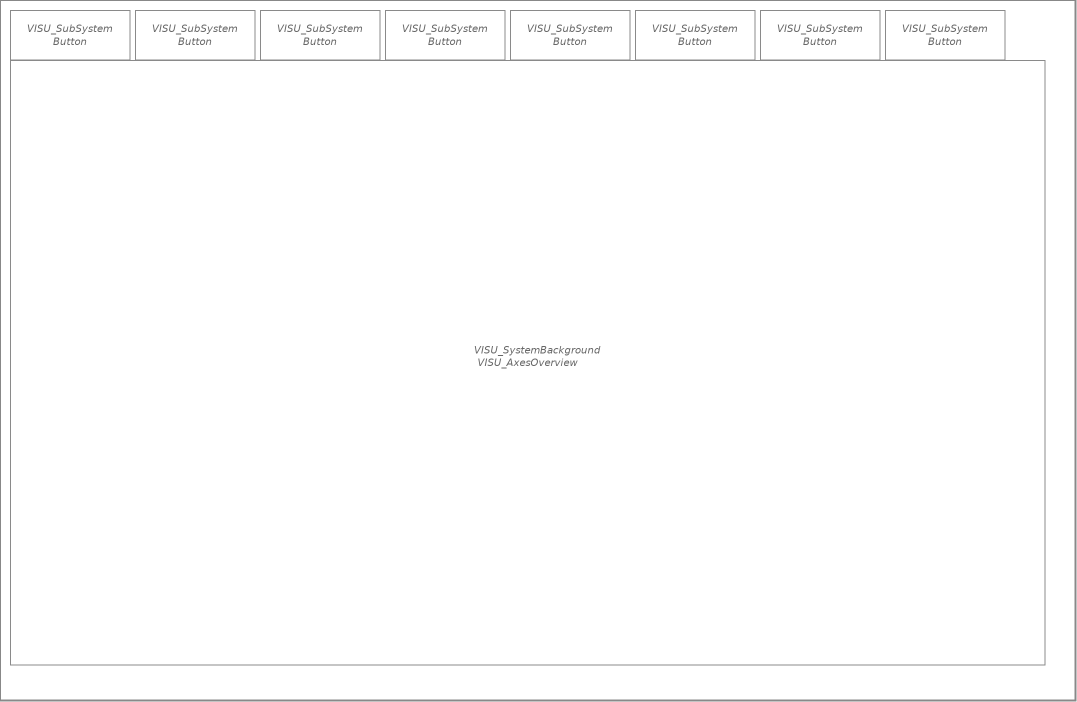
VISUALIZATION VISU_Axes  // 1077x702
VAR_IN_OUT
	ref : Axes;
    widget : AxesWidget;
END_VAR
    Frame (0,0 1075x700)
        shows VISU_SystemBackground(color := widget.actualStatus.color)
    Frame (10,60 1035x605)
        shows VISU_AxesOverview(ref := ref, widget := widget)
        shows VISU_AxesManual(ref := ref, widget := widget.manual)
        shows VISU_AxesAxes(ref := ref, widget := widget.axes)
        shows VISU_AxesTarget(ref := ref, widget := widget)
        shows VISU_AxesPointingModelsSetup(ref := ref.parts.tpoint, widget := widget.tpoint)
        shows VISU_AxesAdvanced(ref := ref, widget := widget)
        shows VISU_AxesIO(ref := ref.parts.io, widget := widget.io)
        shows VISU_AxesConfig(editable := ref.editableConfig, active := ref.config, mgr := ref.parts.configManager, mgrWidget := widget.configManager, axesWidget := widget)
        p701045219: ref.editableConfig
        p2690442461: ref.config
        p942769723: ref.parts.configManager
        p2963374678: widget.configManager
        p459268616: widget
        p4094514409: widget
        p1371549466: ref.editableConfig
        p1340763843: ref.config
        p2803088772: widget
        p2427492753: ref.parts.aziDrive
        p1656878407: ref.parts.ablDrive
        p2190985393: ref.parts.eleDrive
    Frame (10,10 120x50)
        shows VISU_SubSystemButton(widget := widget.button_overview)
        OnMouseClick: FrameSelectionChange Selection=SelectedFrame=b1e9e4b0-bf3d-440f-90c5-cb513105ccf1, GlobSel=AssignType=Directly, SelType=Locally
        OnMouseClick: execute { widget.activeTab := AxesTabs.OVERVIEW; }
    Frame (635,10 120x50)
        shows VISU_SubSystemButton(widget := widget.button_advanced)
        OnMouseClick: FrameSelectionChange Selection=SelectedFrame=b1e9e4b0-bf3d-440f-90c5-cb513105ccf1, Selection=5, GlobSel=AssignType=Directly, SelType=Locally
        OnMouseClick: execute { widget.activeTab := AxesTabs.ADVANCED; }
    Frame (760,10 120x50)
        shows VISU_SubSystemButton(widget := widget.button_io)
        OnMouseClick: FrameSelectionChange Selection=SelectedFrame=b1e9e4b0-bf3d-440f-90c5-cb513105ccf1, Selection=6, GlobSel=AssignType=Directly, SelType=Locally
        OnMouseClick: execute { widget.activeTab := AxesTabs.IO; }
    Frame (135,10 120x50)
        shows VISU_SubSystemButton(widget := widget.button_manual)
        OnMouseClick: FrameSelectionChange Selection=SelectedFrame=b1e9e4b0-bf3d-440f-90c5-cb513105ccf1, Selection=1, GlobSel=AssignType=Directly, SelType=Locally
        OnMouseClick: execute { widget.activeTab := AxesTabs.MANUAL; }
    Frame (260,10 120x50)
        shows VISU_SubSystemButton(widget := widget.button_axes)
        OnMouseClick: FrameSelectionChange Selection=SelectedFrame=b1e9e4b0-bf3d-440f-90c5-cb513105ccf1, Selection=2, GlobSel=AssignType=Directly, SelType=Locally
        OnMouseClick: execute { widget.activeTab := AxesTabs.AXES; }
    Frame (385,10 120x50)
        shows VISU_SubSystemButton(widget := widget.button_target)
        OnMouseClick: FrameSelectionChange Selection=SelectedFrame=b1e9e4b0-bf3d-440f-90c5-cb513105ccf1, Selection=3, GlobSel=AssignType=Directly, SelType=Locally
        OnMouseClick: execute { widget.activeTab := AxesTabs.TARGET; }
    Frame (510,10 120x50)
        shows VISU_SubSystemButton(widget := widget.button_tpoint)
        OnMouseClick: FrameSelectionChange Selection=SelectedFrame=b1e9e4b0-bf3d-440f-90c5-cb513105ccf1, Selection=4, GlobSel=AssignType=Directly, SelType=Locally
        OnMouseClick: execute { widget.activeTab := AxesTabs.TPOINT; }
    Frame (885,10 120x50)
        shows VISU_SubSystemButton(widget := widget.button_config)
        OnMouseClick: FrameSelectionChange Selection=SelectedFrame=b1e9e4b0-bf3d-440f-90c5-cb513105ccf1, Selection=7, GlobSel=AssignType=Directly, SelType=Locally
        OnMouseClick: execute { widget.activeTab := AxesTabs.CONFIG; }
END_VISUALIZATION

(* stored: Version 1.1.0.1, ProductVersion 3.1.4019.2
   Visu VISU_Axes: Id {f8b5a857-8f0c-4e98-86ca-f9d82e0ebe68} *)
